// Core §6.1 — single derived command/module state
{attribute 'qualified_only'}
TYPE E_ExecState :
(
    READY   := 0,
    BUSY    := 1,
    DONE    := 2,
    ERROR   := 3,
    ABORTED := 4
) DINT;
END_TYPE

(* stored: Version 1.1.0.1, ProductVersion 3.1.4024.12
   DUT E_ExecState: Id {170dce39-3bea-48c6-a287-7cd187489385} *)
